{attribute 'qualified_only'}
TYPE E_DistributionType :
(
	Uniform := 0,
	Normal,
	Chi_squared,
	Exponential,
	Gamma
);
END_TYPE

(* stored: Version 1.1.0.1, ProductVersion 3.1.4022.12
   DUT E_DistributionType: Id {1b39f8fe-612a-4136-bde0-715b56490972} *)
